Staubli VAL3: setWordAt.pgx

public program setWordAt(num x_nByteIndex, num x_nWord, num& x_nBuffer[])
  local num l_nHIword
  local num l_nLOword
  local string l_sBinWord
  local string l_sTempBinByte
begin

  //Header begin

  // This function set to "x_nWord" the value of the word composed by two bytes starting from "x_nByteIndex" element of the array x_nBuffer (most likely a plc's memory area we are about to write with writeArea).
  // This will be done according to the Big Endian notation used in Siemens.
  //
  //Input parameters
  //
  //num x_nByteIndex: the index of the element in the "x_nBuffer[]" array representing the starting byte of the word we want to read.
	//num x_nRes: the word value we want to set.
  //
  //Output parameters
  //
  //num x_nBuffer[1]: the monodimensional array of num where we are writing a word (most likely a plc's memory area we are about to write with writeArea).
  //
  //Examples
  //
  // call setWordAt(0,554,l_nLocalWord)
  //
  //History
  // Creation: 24-12-16 - Alessio Villa
  //Header end

  //gestione del segno???
  if x_nWord<0 or x_nWord>power(2,16)-1
    x_nBuffer[x_nByteIndex]=0
    x_nBuffer[x_nByteIndex+1]=0
    return
  endIf

  l_sBinWord=""
  call bitOp:BitWord(x_nWord,l_sBinWord)
  call bitOp:shiftRight(l_sBinWord,8)
  call bitOp:BinToDec(l_sBinWord,l_nLOword)

  l_sBinWord=""
  call bitOp:BitWord(x_nWord,l_sBinWord)
  call bitOp:boolAnd(l_sBinWord,"0000000011111111",l_sTempBinByte)
  call bitOp:BinToDec(l_sTempBinByte,l_nHIword)

  x_nBuffer[x_nByteIndex]=l_nLOword
  x_nBuffer[x_nByteIndex+1]=l_nHIword

end
